FUNCTION_BLOCK abstract FB_UniversalVFDModbus EXTENDS FB_ModbusSlave IMPLEMENTS I_UniversalVFD
VAR
	eVfdState	: E_Vfd_State;
	bInit	: BOOL;
	bBusy	: BOOL;
	bReset	: BOOL;
	bStop	: BOOL;
	bAbort : BOOL;
	bError : BOOL;
	bWarning : BOOL;// status
	bRunningForward	: BOOL;// in state running forward
	bRunningReverse	: BOOL; // in state running reverse
	bRanForward	: BOOL;
	bRanReverse	: BOOL;
	lrHzActual	: LREAL;
	lrDcVoltage		: LREAL;
	lrVacOutToMotor	: LREAL;
	lrCurrent	: LREAL;	
	lrPowerKw	: LREAL;	
	eVfdStatus	: E_VFD_Status;
	lrHzControl	: LREAL;// value in range(0.0-50.0Hz)
	iErrorID		: UDINT;

	lrSpeed : LREAL;
	lrTorque : LREAL;
	lrTotalKwh : LREAL;
	lrRatedPower : LREAL;
	bActive: BOOL;
	bOverLoad: BOOL;
	bStopLog: BOOL;
	bStopped: BOOL;
	
	VFD_CTRL_RESET_FAULT : WORD;
	VFD_CTRL_RUN_FORWARD :WORD;
	VFD_CTRL_RUN_REVERSE :WORD ;
	VFD_CTRL_STOP_FREE 		:WORD ;
	VFD_CTRL_STOP_SPEED_DOWN	:WORD ;
	
	tonStopDelay: Ton;
	// time delay after status = stop
	tStopDelay: TIME := T#4S;
	bReallyError	: BOOL;// because of bError maybe incorrect because noise information return by Modbus
	tonConfirmReallyError : TON;
	timeConfirmReallyError : TIME := T#15S;
END_VAR
VAR CONSTANT
	// index
	iCTRL_WORD	: UINT := 1;
	iCTRL_FREQUENCY_WORD :UINT := 0;
	iSTATUS_WORD	: UINT := 0;
END_VAR

StateMachine();
CASE eVfdStatus OF
	VFD_STATUS_RUNNING_FORWARD :
		bRanForward := TRUE;
		bRanReverse := FALSE;
		bStopped := FALSE;
	VFD_STATUS_RUNNING_REVERSE:
		bRanForward := FALSE;
		bRanReverse := TRUE;
		bStopped := FALSE;
	VFD_STATUS_FAULT,VFD_STATUS_STOP:
		bRanForward := FALSE;
		bRanReverse := FALSE;
		bStopped := TRUE;
		
END_CASE
bError := eVfdStatus = VFD_STATUS_FAULT;
bActive := eVfdState >= VFD_IDLE;
CASE eVfdState OF
	VFD_INITIALIZING..VFD_RESET_DONE, VFD_ABORTING:
		tonConfirmReallyError(
			IN := bError OR iModbusErrorID <> MODBUSERROR_NO_ERROR,
			PT := timeConfirmReallyError,
			Q => bReallyError 
		);
END_CASE

{attribute 'monitoring' := 'variable'}
PROPERTY Active : REFERENCE TO  bool
GET
Active REF= bActive;
END_GET
END_PROPERTY

PROPERTY AcVoltageToMotor : Reference to lreal
GET
AcVoltageToMotor ref= lrVacOutToMotor;
END_GET
END_PROPERTY

{attribute 'monitoring' := 'variable'}
PROPERTY Busy : reference to bool
GET
Busy ref= bBusy;
END_GET
END_PROPERTY

METHOD Convert : BOOL
VAR_INPUT
	iRegionNo	:	INT;
	pReadData	:	POINTER TO word;
END_VAR
(*CASE iRegionNo OF
	0:
		// Status word
		Inverter_Ready		:=  pReadData[0].0;
		InverterReadyToRun	:=  pReadData[0].1;
		InverterRunning		:=  pReadData[0].2;
		InverterFaultActive :=  pReadData[0].3;
		OFF2_active			:= NOT pReadData[0].4;
		OFF3_active			:= NOT  pReadData[0].5;
		ON_inhibit_active 	 := pReadData[0].6;
		Inverter_warning_active := pReadData[0].7;
		Deviation_setpoint_OR_ActiveValue := NOT pReadData[0].8;
		PZD_control 		:= pReadData[0].9;
		Motor_current_Or_torque_limit  := NOT pReadData[0].11;
		Brake_open	 := pReadData[0].12;
		Motor_overload := NOT pReadData[0].13;
		Motor_RunRight	:= pReadData[0].14;
		Inverter_overload :=  NOT pReadData[0].15;
		
		IF InverterFaultActive THEN
			eStatus := VFD_STATUS_FAULT;
		ELSIF InverterFaultActive THEN
			eStatus := VFD_STATUS_WARNING;
		ELSIF InverterRunning THEN
			IF Motor_RunRight THEN
				eStatus := VFD_STATUS_RUNNING_FORWARD;
			ELSE
				eStatus := VFD_STATUS_RUNNING_REVERSE;
			END_IF
		ELSIF NOT InverterRunning THEN
			eStatus := VFD_STATUS_STOP;
		END_IF

		// Speed word
		lrHz_actual := WORD_TO_LREAL( pReadData[1])*50/16383;
		
	1:
		///  actual  Speed ( rpm) (unit A : Scale factor 1), Current ( A , 100, , Torque (Nm, 100)
	//, Actual Power (kw, 100), Total Kwh( 1), Dc bus Voltage(1), REFERENCE( hz, 100), RATED PWR( 100),OUTPUT VOLTS(1)
		lrSpeed := pReadData[0];
		lrCurrent := WORD_TO_LREAL(pReadData[1])/100;
		lrTorque := WORD_TO_LREAL(pReadData[2])/100;
		lrPower := WORD_TO_LREAL(pReadData[3])/100;
		lrTotalKwh := WORD_TO_LREAL(pReadData[4]);
		lrDc_Voltage := WORD_TO_LREAL(pReadData[5]);
		lrRatedPower := WORD_TO_LREAL(pReadData[7])/100;
		lrVAC_OutToMotor := WORD_TO_LREAL(pReadData[8]);
END_CASE
*)
END_METHOD

PROPERTY Current : reference to lreal
GET
Current ref= lrCurrent;
END_GET
END_PROPERTY

PROPERTY DcVoltage : Reference to lreal
GET
DcVoltage ref= lrDcVoltage;
END_GET
END_PROPERTY

{attribute 'monitoring' := 'variable'}
PROPERTY Error : REFERENCE to bool
GET
Error ref= bError;
END_GET
END_PROPERTY

{attribute 'monitoring' := 'variable'}
PROPERTY ErrorID : reference to UDINT
GET
ErrorID ref= iErrorID;
END_GET
END_PROPERTY

METHOD  FirstCycle 
VAR_INPUT
	sName : STRING;
	iUnitID : BYTE ; // modbus address of the device : 1- 255
END_VAR
THIS^.sName := sName;
THIS^.iUnitID := iUnitID;
(*(*HSW (speed setpoint), HIW (actual speed), STW (control word), ZSW (status word) refer to
control data. For more information, see parameters r2018 and P2019 in Chapter "Parameter
list (Page 147)*)
//ZSW  (status WORD), HIW (actual speed)
	arrAddress[0][0] := 109;
	arrAddress[0][1]	:= 2;

///  actual  Speed ( rpm) (unit A : Scale factor 1), Current ( A , 100, , Torque (Nm, 100)
	//, Actual Power (kw, 100), Total Kwh( 1), Dc bus Voltage(1), REFERENCE( hz, 100), RATED PWR( 100),OUTPUT VOLTS(1)
	arrAddress[1][0] := 24;
	arrAddress[1][1] := 10;

	
iNumAddRegion	:= 2;
/////write control  VFD
	
// Frequency

arrAddressWrite[0][0]	:= 100;
arrAddressWrite[0][1] 	:= 1;
arrAddressWrite[0][2]	:= LREAL_TO_WORD( FC_ScaleValue(	rangeRawMin := 0,
															rangeRawMax := 50,
															RangeScaleMin :=0,
															RangeScaleMax := 16384,
															ValueRaw := lrHz_Control) );
// Control word																	
arrAddressWrite[1][0]	:= 99;
arrAddressWrite[1][1] := 1;
arrAddressWrite[1][2]	:= 1150; //VFD_CTRL_STOP_SPEED_DOWN
iNumAddRegionWrite := 2;
*)
END_METHOD

PROPERTY HzActual : REFERENCE TO  LReal
GET
HzActual ref= lrHzActual;
END_GET
END_PROPERTY

PROPERTY HzControl : reference to LReal
GET
HzControl ref= lrHzControl;
END_GET
END_PROPERTY

{attribute 'monitoring' := 'variable'}
PROPERTY InHz : bool
GET
InHz :=  FC_InRange( bound1 := lrHzControl +1,
					bound2 := lrHzControl -1,
					value := lrHzActual) ;
END_GET
END_PROPERTY

PROPERTY isRunForward : bool
GET
isRunForward := bRanForward;
END_GET
END_PROPERTY

{attribute 'monitoring' := 'variable'}
PROPERTY IsRunning : bool
GET
IsRunning := eVfdStatus = VFD_STATUS_RUNNING_FORWARD
			 OR  eVfdStatus = VFD_STATUS_RUNNING_REVERSE;
END_GET
END_PROPERTY

PROPERTY isRunReverse : bool
GET
isRunReverse := bRanReverse;
END_GET
END_PROPERTY

PROPERTY isStop : bool
GET
isStop := bStopped;
END_GET
END_PROPERTY

METHOD MR_Abort : BOOL
VAR_INPUT
END_VAR
IF eVfdState >= VFD_INITIALIZING THEN
	bAbort := TRUE;
	eVfdState := VFD_ABORTING;
	fbMachineLogger.MR_AddLogs(CONCAT(sName,' : abort requested'));
	bBusy := TRUE;
	
ELSIF eVfdState = VFD_UNINITIALIZED THEN
	bAbort 		:= FALSE;
	MR_Abort	:= TRUE;
	bBusy := FALSE;
	fbMachineLogger.MR_AddLogs(CONCAT(sName,' : abort done'));
	
END_IF
END_METHOD

METHOD MR_Init : bool
VAR_INPUT
END_VAR
IF eVFDState = VFD_UNINITIALIZED THEN
	bInit := TRUE;
	MR_Init := FALSE;
	eVfdState := VFD_INITIALIZING;
	fbMachineLogger.MR_AddLogs(CONCAT(sName,' : initialization requested'));
	bBusy := TRUE;
	
ELSIF eVFDState = VFD_READY_INITIALIZED THEN
	bInit := FALSE;
	MR_Init := TRUE;
	bBusy := FALSE;
	fbMachineLogger.MR_AddLogs(CONCAT(sName,' : initialization done'));
END_IF
END_METHOD

METHOD MR_Reset : BOOL
VAR_INPUT
END_VAR
IF eVfdState >= VFD_IDLE AND bError THEN
	bReset := TRUE;
	eVfdState := VFD_RESET;
	fbMachineLogger.MR_AddLogs(CONCAT(sName,' : reset requested'));			
	bBusy := TRUE;
	
ELSIF eVfdState = VFD_RESET_DONE THEN
	bError := FALSE;
	iErrorID := 0;
	bReset := FALSE;
	MR_Reset := TRUE;
	bBusy := FALSE;
	fbMachineLogger.MR_AddLogs(CONCAT(sName,' : reset done'));		
		
END_IF
END_METHOD

METHOD MR_RunForward : BOOL
VAR_INPUT
	hz : LREAL; 
END_VAR
IF eVfdState = VFD_IDLE  AND (NOT  FC_InRange( 	bound1 := lrHzControl + 0.01,
												bound2 := lrHzControl - 0.01,
												value :=  hz)
								OR bRanReverse
								OR bStopped)
THEN
	lrHzControl := hz;
	bRunningForward := TRUE;
	MR_RunForward := FALSE;
	eVfdState := VFD_RUN_FORWARD;
	fbMachineLogger.MR_AddLogs( sLogMessage := FUN_MergeStrings4(  sName,' : run ',LREAL_TO_STRING( lrHzControl),' forward requested'));		
	bBusy := TRUE;
	
ELSIF eVfdState = VFD_RUN_FORWARD_DONE THEN
	bRunningForward := FALSE;
	MR_RunForward := TRUE;
	fbMachineLogger.MR_AddLogs(CONCAT(sName,' : run forward done'));	
	bBusy := FALSE;
END_IF
END_METHOD

METHOD MR_RunReverse : BOOL// must stop before call run reverse or forward
VAR_INPUT
	hz : LREAL; // >0 and < 50;
END_VAR
IF eVfdState = VFD_IDLE  AND (NOT  FC_InRange( 	bound1 := lrHzControl + 0.01,
												bound2 := lrHzControl - 0.01,
												value :=  hz)
								OR bRanForward
								OR bStopped)
THEN
	lrHzControl := hz;
	bRunningReverse := TRUE;
	MR_RunReverse := FALSE;
	eVfdState := VFD_RUN_REVERSE;
	fbMachineLogger.MR_AddLogs( sLogMessage := FUN_MergeStrings4(  sName,' : run ',LREAL_TO_STRING( lrHzControl),' forward requested'));		
	bBusy := TRUE;
	
ELSIF eVfdState = VFD_RUN_REVERSE_DONE THEN
	bRunningReverse := FALSE;
	MR_RunReverse := TRUE;
	fbMachineLogger.MR_AddLogs(CONCAT(sName,' : run forward done'));
	bBusy := FALSE;
END_IF
END_METHOD

METHOD MR_Stop : BOOL
VAR_INPUT
END_VAR
IF eVfdState >= VFD_IDLE AND eVfdState <> VFD_STOP_DONE THEN
	IF NOT bStopLog THEN 
		fbMachineLogger.MR_AddLogs(CONCAT(sName,' : stop requested'));
		bStopLog := TRUE;	
	END_IF
	
	bStop := TRUE;
	eVfdState := VFD_STOP;
	bBusy := TRUE;
	
ELSIF eVfdState = VFD_STOP_DONE THEN
	bStop 		:= FALSE;
	MR_Stop 	:= TRUE;
	bStopLog 	:= FALSE;
	fbMachineLogger.MR_AddLogs(CONCAT(sName,' : stop done'));	
	bBusy := FALSE;
END_IF
END_METHOD

METHOD PROTECTED MS_Aborting
lrHzControl := 0;
bInit := FALSE;
bRunningForward := FALSE;
bRunningReverse := FALSE;
bReset := FALSE;
bRanForward := FALSE;
bRanReverse := FALSE;
bOverLoad := FALSE;
bStop := FALSE;
bStopLog := FALSE;
bStopped := FALSE;
THIS^.tonStopDelay(IN :=FALSE);
IF eVfdStatus = VFD_STATUS_STOP OR eVfdStatus = VFD_STATUS_FAULT THEN
	eVfdState := VFD_UNINITIALIZED;
END_IF
END_METHOD

METHOD PROTECTED MS_Idle
;
END_METHOD

METHOD  PROTECTED  MS_Initializing
// from Subclass call Super^.MS_Initializing
arrAddressWrite[iCTRL_WORD][2]	:= VFD_CTRL_RESET_FAULT;
IF eVfdStatus = VFD_STATUS_READY_TO_RUN THEN
	eVFDState := VFD_READY_INITIALIZED;
END_IF
END_METHOD

METHOD PROTECTED MS_ReadyInitialized
VAR_INPUT
END_VAR
IF NOT bInit THEN
	eVfdState := VFD_IDLE;
END_IF
END_METHOD

METHOD PROTECTED  MS_Reset
VAR_INPUT
END_VAR
arrAddressWrite[iCTRL_WORD][2]	:= VFD_CTRL_RESET_FAULT;
IF THIS^.evfdStatus <>  VFD_STATUS_NOT_RESPOND AND
	THIS^.evfdStatus <>  VFD_STATUS_FAULT THEN
	evfdState := VFD_RESET_DONE;
END_IF
END_METHOD

METHOD PROTECTED MS_ResetDone
VAR_INPUT
END_VAR
IF NOT bReset THEN
	evfdState := VFD_IDLE;
END_IF
END_METHOD

METHOD PROTECTED  MS_RunForward
VAR_INPUT
END_VAR
(*arrAddressWrite[iCtrlFrequencyWord][2] :=  LREAL_TO_WORD( 
											FC_ScaleValue(		rangeRawMin := 0,
																rangeRawMax := 50,
																RangeScaleMin := WORD_TO_LREAL( wHzWordValueMin),
																RangeScaleMax := WORD_TO_LREAL( wHzWordValueMax),
																ValueRaw := lrHzControl) 
														);*)
arrAddressWrite[iCTRL_WORD][2]	:= VFD_CTRL_RUN_FORWARD;
IF eVfdStatus = VFD_STATUS_RUNNING_FORWARD 
(*AND F_InRange( bound1 := lrHzControl + 1,
				bound2 := lrHzControl -1,
				value := lrHzActual)*)
THEN
	eVFDState := VFD_RUN_FORWARD_DONE;
END_IF
END_METHOD

METHOD PROTECTED MS_RunForwardDone
IF NOT bRunningForward THEN
	eVfdState := VFD_IDLE;
END_IF
END_METHOD

METHOD PROTECTED  MS_RunReverse
VAR_INPUT
END_VAR
(*arrAddressWrite[iCtrlFrequencyWord][2] :=  LREAL_TO_WORD( 
											FC_ScaleValue(		rangeRawMin := 0,
																rangeRawMax := 50,
																RangeScaleMin := WORD_TO_LREAL( wHzWordValueMin),
																RangeScaleMax := WORD_TO_LREAL( wHzWordValueMax),
																ValueRaw := lrHzControl) 
														);*)
arrAddressWrite[iCTRL_WORD][2]	:= VFD_CTRL_RUN_REVERSE;
IF eVfdStatus = VFD_STATUS_RUNNING_REVERSE 
(*AND F_InRange( bound1 := lrHzControl + 1,
				bound2 := lrHzControl -1,
				value := lrHzActual)*)
THEN
	eVFDState := VFD_RUN_REVERSE_DONE;
END_IF
END_METHOD

METHOD PROTECTED MS_RunReverseDone
VAR_INPUT
END_VAR
IF NOT bRunningReverse THEN
	eVfdState := VFD_IDLE;
END_IF
END_METHOD

METHOD protected  MS_Stop 
VAR_INPUT
END_VAR
arrAddressWrite[iCTRL_WORD][2]	:= VFD_CTRL_STOP_SPEED_DOWN;
(*tonStopDelay( in := eVfdStatus = VFD_STATUS_STOP,
				PT := tStopDelay);*)
IF eVfdStatus = VFD_STATUS_STOP THEN
 eVfdState := VFD_STOP_DONE;	
END_IF
(*IF tonStopDelay.Q THEN
	tonStopDelay(IN := FALSE);
	
END_IF*)
END_METHOD

METHOD protected Ms_StopDone
VAR_INPUT
END_VAR
IF NOT bStop THEN
	eVfdState := VFD_IDLE;
END_IF
END_METHOD

METHOD PROTECTED MS_Uninitialized
END_METHOD

{attribute 'monitoring' := 'variable'}
PROPERTY Overload : reference TO BOOL
GET
Overload REF= bOverLoad;
END_GET
END_PROPERTY

{attribute 'monitoring' := 'variable'}
PROPERTY PowerKw : REFERENCE TO LREAL
GET
PowerKw ref= lrPowerKw;
END_GET
END_PROPERTY

PROPERTY ReallyError : bool
GET
ReallyError := bReallyError;
END_GET
END_PROPERTY

PROPERTY Speed : Reference to lreal
GET
Speed REF= lrSpeed;
END_GET
END_PROPERTY

{attribute 'monitoring' := 'variable'}
PROPERTY State : reference to E_Vfd_State
GET
State REF= eVfdState;
END_GET
END_PROPERTY

METHOD PROTECTED StateMachine
CASE eVfdState OF
	VFD_UNINITIALIZED :
		MS_Uninitialized();
		
	VFD_INITIALIZING	:
		MS_Initializing();
		
	VFD_READY_INITIALIZED :
		MS_ReadyInitialized();
		
	VFD_IDLE:
		MS_Idle();
	
	VFD_RUN_FORWARD	:
		MS_RunForward();
		
	VFD_RUN_FORWARD_DONE:
		MS_RunForwardDone();
	
	VFD_RUN_REVERSE	:
		MS_RunReverse();
	
	VFD_RUN_REVERSE_DONE:
		MS_RunReverseDone();
	
	VFD_STOP		:
		MS_Stop();
		
	VFD_STOP_DONE	:
		Ms_StopDone();
		
	VFD_RESET	:
		MS_Reset();
		
	VFD_RESET_DONE	:
		MS_ResetDone();
		
	VFD_ABORTING :
		MS_Aborting();
	
	
END_CASE
END_METHOD

{attribute 'monitoring' := 'variable'}
PROPERTY Status : reference to E_VFD_Status
GET
Status REF= eVfdStatus;
END_GET
END_PROPERTY

PROPERTY TimeRemainConfirmReallyError : Time
GET
TimeRemainConfirmReallyError := timeConfirmReallyError;
END_GET
SET
timeConfirmReallyError := TimeRemainConfirmReallyError;
END_SET
END_PROPERTY

PROPERTY timeStopDelay : time
GET
timeStopDelay := THIS^.tStopDelay;
END_GET
SET
tStopDelay := timeStopDelay;
END_SET
END_PROPERTY

PROPERTY Torque : reference to lreal
GET
Torque ref= Torque;
END_GET
END_PROPERTY

PROPERTY TotalKwh : reference to lreal
GET
TotalKwh REF= TotalKwh;
END_GET
END_PROPERTY

// not all vfd modbus available this function 
PROPERTY Warning : reference to bool
GET
Warning  ref= bWarning;
END_GET
END_PROPERTY

END_FUNCTION_BLOCK

(* stored: Version 1.1.0.1, ProductVersion 3.1.4024.12
   POU FB_UniversalVFDModbus: Id {218756d0-612e-48ed-8e53-949cee63529d}, SpecialFunc None
   Folder MR: Id {bd5cd554-879a-4201-b28f-5c47833969b1}
   Folder MS: Id {c35aa3da-6bb6-415a-8b39-338b5a806a33}
   Folder Pro: Id {445a1ee2-8690-4398-8958-7a1d7b41ed02}
   Property Active: Id {c27887fb-c492-4b7e-89d7-acc86faca04e}
   Get Get: Id {231f04f1-854b-4524-9a7a-30adf2b5b005}
   Property AcVoltageToMotor: Id {5f14a5f9-5f3b-4e73-afd6-4f18bb63ad97}
   Get Get: Id {3ddff3cf-335e-4a44-8f33-79a2c852bd07}
   Property Busy: Id {5c85f589-4485-4bfe-bd13-199f6fff2509}
   Get Get: Id {bd76c115-ffef-4561-b825-e1d3c3825fab}
   Method Convert: Id {f4c08b77-e954-42a5-a631-8c5995d9fc69}
   Property Current: Id {cc7adb18-6008-4197-84ca-4e61116074bf}
   Get Get: Id {f35cc3d5-4da7-4eae-bc5f-44e69aaa95a1}
   Property DcVoltage: Id {53eb5e87-ac44-4e26-bdd8-0ee08e91b7e8}
   Get Get: Id {c683587c-b857-4874-ab4d-db02ef3fbb50}
   Property Error: Id {2bdb6e30-c54b-4bd0-8a8d-de32e855496b}
   Get Get: Id {ef6fe521-bf9a-49fb-bd4b-7a6c9eaf8a3d}
   Property ErrorID: Id {f2add6d4-3cb6-4456-98da-b86715ce6415}
   Get Get: Id {80a17aea-9757-4c00-b6f6-f4afdc019293}
   Method FirstCycle: Id {6d68d29c-2866-4975-9c45-ac338928650a}
   Property HzActual: Id {a63535e9-b079-49cc-8cfa-02bbf8cb6d1e}
   Get Get: Id {cd46b4cf-0fb4-440e-b73f-acf8eb29658f}
   Property HzControl: Id {847818af-6a3e-419c-8ee5-51bdc748b99a}
   Get Get: Id {260d3f56-0967-483d-adb3-80d29413a8b1}
   Property InHz: Id {0973b887-90fc-413b-bd37-5bf992843711}
   Get Get: Id {69d3d820-32e7-45d3-a12b-d1a3933ffc71}
   Property isRunForward: Id {4e8709e3-c3da-4223-bf00-223409f23591}
   Get Get: Id {64d7e920-73d1-4775-8289-b6df3e8537d2}
   Property IsRunning: Id {57e0a5a9-5b9d-4c3d-93e8-4b7cf5aec1f5}
   Get Get: Id {80f9fef0-6bb9-43ac-8927-635f16841f31}
   Property isRunReverse: Id {5fbf05b3-6f19-49f6-86e2-daff83e0df6c}
   Get Get: Id {9642e99e-b93c-471e-9b49-28795e09f6f9}
   Property isStop: Id {86232ba9-ab3b-4cf0-9c96-041239f4c168}
   Get Get: Id {6cf5cf41-ff30-4216-b1e7-d5771894c0b4}
   Method MR_Abort: Id {e8a80b2d-2673-4346-a00d-c0d102e5c82d}
   Method MR_Init: Id {de2a3891-47d3-4163-a868-ce0528202b5e}
   Method MR_Reset: Id {2bdc3e6e-4954-4190-9f28-8a8457e364d7}
   Method MR_RunForward: Id {db4982e0-0c38-4a5a-b38a-2adf1fd682c3}
   Method MR_RunReverse: Id {35569046-4001-4b47-8999-0c6321e7807c}
   Method MR_Stop: Id {d61e11cb-90ac-46df-8a8d-2188731f7dcc}
   Method MS_Aborting: Id {7340f979-e913-4927-813d-53316372cb0e}
   Method MS_Idle: Id {1ee53fd3-372d-4672-9b04-0f6ce059bbab}
   Method MS_Initializing: Id {04d14cc6-499b-4615-ae1c-95f29a3150f2}
   Method MS_ReadyInitialized: Id {58d13ab0-a73a-4623-ae39-146cb94f2b60}
   Method MS_Reset: Id {298ba71e-5369-4756-8847-56a792cfe08b}
   Method MS_ResetDone: Id {4df641f5-7b99-4d14-97cc-206423cbaaff}
   Method MS_RunForward: Id {9bbcb090-e2cf-49e5-aaa9-3d67622499d4}
   Method MS_RunForwardDone: Id {0e3b2cbb-907c-4c66-b746-e97509edbba3}
   Method MS_RunReverse: Id {aa6997a8-d244-4c31-b7b3-b93d881f69d3}
   Method MS_RunReverseDone: Id {666b33b6-f7e3-46b4-b41e-b130ccc3d405}
   Method MS_Stop: Id {4d46d6c7-2573-43e9-b4a6-e57c14b29b10}
   Method Ms_StopDone: Id {ec169d85-a240-4686-9bf3-b74eadf19895}
   Method MS_Uninitialized: Id {3d98b249-ea9d-4787-81b3-3aaa1d95c98a}
   Property Overload: Id {344fd9fe-f321-4c65-826f-14cbdf07507d}
   Get Get: Id {96d199ff-e553-4442-860f-f94594a6a7f1}
   Property PowerKw: Id {80c7f671-fa73-4d38-bd04-d083dea8ea36}
   Get Get: Id {45caf024-a6be-4331-b374-785a09f8350e}
   Property ReallyError: Id {8e2b83e0-76bb-4f3e-97d7-7866642c71e2}
   Get Get: Id {e3707793-3c28-4420-8b34-6606cfefdc39}
   Property Speed: Id {753ba39a-41cb-4b72-9fe3-f3313de28591}
   Get Get: Id {49930f98-2860-4343-85f5-4283bd6231b6}
   Property State: Id {071f044c-ec91-4cc5-b4f4-08633519aa8a}
   Get Get: Id {8e514446-450b-4a10-82c2-8bbac004b178}
   Method StateMachine: Id {06e5e80d-790e-4127-8b0c-077bc3b579df}
   Property Status: Id {369fec46-0056-41ca-87a6-cdc0cadd1ea3}
   Get Get: Id {9e4eee11-2bc6-4f05-ae9a-2813c54f5019}
   Property TimeRemainConfirmReallyError: Id {97227d1d-9ac2-479c-b8b9-de2e13922015}
   Get Get: Id {c2187032-d548-43f8-abc8-7698e3a6ff53}
   Set Set: Id {dc86321d-4dc3-4b75-8f15-b97a6865b9ae}
   Property timeStopDelay: Id {bddd152c-7479-48f5-a66d-6af59f3be079}
   Get Get: Id {6ed82530-9480-4aa9-98cf-49da6417bb21}
   Set Set: Id {27b9ddbc-8f22-48ee-a23d-b9c5730d0081}
   Property Torque: Id {3d53aa45-cc32-4e2d-a6b4-ef840ef74b12}
   Get Get: Id {799b82bf-dc00-41b0-bd11-9b01342aa577}
   Property TotalKwh: Id {ec495c03-f67d-4bb0-89a4-4d9fcde617e4}
   Get Get: Id {c9add1a0-2dcc-4a63-869c-c84bcfb97d64}
   Property Warning: Id {093b7dd2-48f2-40e7-9e74-deed0479d751}
   Get Get: Id {6add1c7d-ca63-4792-9026-eccda019afad} *)
